REGION Network 37: [Spare_3] valve logic
   // Setup  //  Parametrierungshinweise
   // I_OpModeOutput  -->
   // 0=I_AutoOn schaltet den Ausgang Ein und Aus; 1=I_AutoOn schaltet ein und I_AutoAus schaltet aus
   // 0=I_AutoOn switches on and off; 1=I_AutoOn switches on and I_AutoOff switches off
   // 
   // I_OpModeAutoManual -->
   // 0=Automatik; 1=Hand
   // 0=Automatic; 1=Manual
   // 
   // I_AutoOn -->
   // 1=Automatik Ein, Eingang für die normalen Ventilverschaltungsbedingungen
   // 1=Automatic On, Input for the normal valve conditions
   // 
   // I_Release -->
   // 1=Freigabe, Eingang für die Fehlerbedingungen
   // 1=Release, Input for fault conditions
   // 
   // I_SafetyRelease -->
   // 1=Sicherheitsfreigabe, Eingang für zusätzliche Schaltbefehle aus dem Sicherheitsprogramm
   // 1=Safety release, Input for additional safety conditions from the safety program
   RUNG wire#powerrail
      Move(in := 0, out1 => "DB_R134a_BU_Values".Valve.Spare_3.Input.OpModeOutput)
      Move(in := "DB_R134a_AT_2_Values".OperationMode.ManualValveControl, out1 => "DB_R134a_BU_Values".Valve.Spare_3.Input.OpModeAutoManual)
      { S7_Templates := "SrcType := Int" } EQ_Contact(in1 := "DB_R134a_BU_Values".Valve.Spare_3.Input.OpModeAutoManual, in2 := 0)
      R_Coil( "DB_R134a_BU_Values".Valve.Spare_3.Input.ManualOn )
   END_RUNG
   RUNG wire#powerrail
      Contact( #Tmp_EnableOperation )
      Contact( "AlwaysFALSE" )
      Coil( "DB_R134a_BU_Values".Valve.Spare_3.Input.AutoOn )
   END_RUNG
   RUNG wire#powerrail
      Coil( "DB_R134a_BU_Values".Valve.Spare_3.Input.Release )
   END_RUNG
   RUNG wire#powerrail
      Coil( "DB_R134a_BU_Values".Valve.Spare_3.Input.SafetyRelease )
   END_RUNG
   RUNG wire#powerrail
      MOVE_BLK_VARIANT(SRC := "DB_R134a_1_StepData".Valve[1].Language, COUNT := 4, SRC_INDEX := 0, DEST_INDEX := 0, Ret_Val => #Tmp_ReturnValue, DEST => "DB_R134a_BU_Values".Valve.Spare_3.Input.TextName_Language)
   END_RUNG
   // the same network as SCL:
   "DB_R134a_BU_Values".Valve.Spare_3.Input.OpModeOutput := 0;
   "DB_R134a_BU_Values".Valve.Spare_3.Input.OpModeAutoManual := "DB_R134a_AT_2_Values".OperationMode.ManualValveControl;
   IF "DB_R134a_BU_Values".Valve.Spare_3.Input.OpModeAutoManual = 0 THEN
       "DB_R134a_BU_Values".Valve.Spare_3.Input.ManualOn := FALSE;
   END_IF;
   "DB_R134a_BU_Values".Valve.Spare_3.Input.AutoOn := #Tmp_EnableOperation AND "AlwaysFALSE";
   "DB_R134a_BU_Values".Valve.Spare_3.Input.Release := TRUE;
   "DB_R134a_BU_Values".Valve.Spare_3.Input.SafetyRelease := TRUE;
   #Tmp_ReturnValue := MOVE_BLK_VARIANT(SRC := "DB_R134a_1_StepData".Valve[1].Language,
                           COUNT := 4,
                           SRC_INDEX := 0,
                           DEST_INDEX := 0,
                           DEST => "DB_R134a_BU_Values".Valve.Spare_3.Input.TextName_Language);
END_REGION

REGION Network 38: [Spare_3] valve 1KM1VI1KKP11KKR14 - xxx.. - spare // Reserve
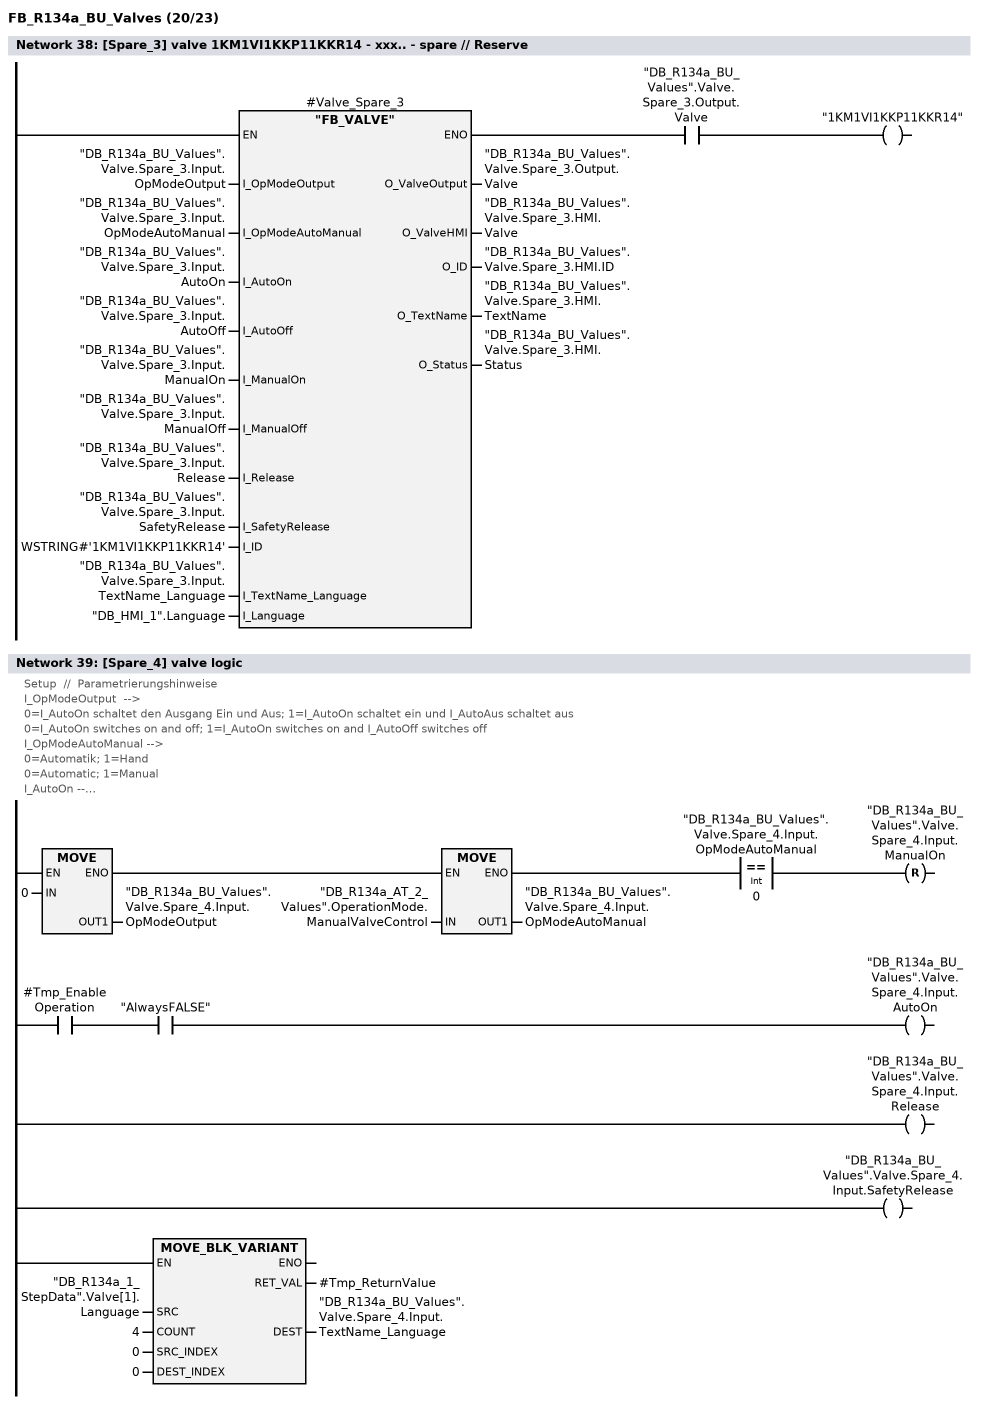
   RUNG wire#powerrail
      #Valve_Spare_3(I_OpModeOutput := "DB_R134a_BU_Values".Valve.Spare_3.Input.OpModeOutput, I_OpModeAutoManual := "DB_R134a_BU_Values".Valve.Spare_3.Input.OpModeAutoManual, I_AutoOn := "DB_R134a_BU_Values".Valve.Spare_3.Input.AutoOn, I_AutoOff := "DB_R134a_BU_Values".Valve.Spare_3.Input.AutoOff, I_ManualOn := "DB_R134a_BU_Values".Valve.Spare_3.Input.ManualOn, I_ManualOff := "DB_R134a_BU_Values".Valve.Spare_3.Input.ManualOff, I_Release := "DB_R134a_BU_Values".Valve.Spare_3.Input.Release, I_SafetyRelease := "DB_R134a_BU_Values".Valve.Spare_3.Input.SafetyRelease, I_ID := WSTRING#'1KM1VI1KKP11KKR14', I_TextName_Language := "DB_R134a_BU_Values".Valve.Spare_3.Input.TextName_Language, I_Language := "DB_HMI_1".Language, O_ValveOutput => "DB_R134a_BU_Values".Valve.Spare_3.Output.Valve, O_ValveHMI => "DB_R134a_BU_Values".Valve.Spare_3.HMI.Valve, O_ID => "DB_R134a_BU_Values".Valve.Spare_3.HMI.ID, O_TextName => "DB_R134a_BU_Values".Valve.Spare_3.HMI.TextName, O_Status => "DB_R134a_BU_Values".Valve.Spare_3.HMI.Status)
      Contact( "DB_R134a_BU_Values".Valve.Spare_3.Output.Valve )
      Coil( "1KM1VI1KKP11KKR14" )
   END_RUNG
   // the same network as SCL:
   #Valve_Spare_3(I_OpModeOutput := "DB_R134a_BU_Values".Valve.Spare_3.Input.OpModeOutput,   // "FB_VALVE"
                  I_OpModeAutoManual := "DB_R134a_BU_Values".Valve.Spare_3.Input.OpModeAutoManual,
                  I_AutoOn := "DB_R134a_BU_Values".Valve.Spare_3.Input.AutoOn,
                  I_AutoOff := "DB_R134a_BU_Values".Valve.Spare_3.Input.AutoOff,
                  I_ManualOn := "DB_R134a_BU_Values".Valve.Spare_3.Input.ManualOn,
                  I_ManualOff := "DB_R134a_BU_Values".Valve.Spare_3.Input.ManualOff,
                  I_Release := "DB_R134a_BU_Values".Valve.Spare_3.Input.Release,
                  I_SafetyRelease := "DB_R134a_BU_Values".Valve.Spare_3.Input.SafetyRelease,
                  I_ID := WSTRING#'1KM1VI1KKP11KKR14',
                  I_TextName_Language := "DB_R134a_BU_Values".Valve.Spare_3.Input.TextName_Language,
                  I_Language := "DB_HMI_1".Language,
                  O_ValveOutput => "DB_R134a_BU_Values".Valve.Spare_3.Output.Valve,
                  O_ValveHMI => "DB_R134a_BU_Values".Valve.Spare_3.HMI.Valve,
                  O_ID => "DB_R134a_BU_Values".Valve.Spare_3.HMI.ID,
                  O_TextName => "DB_R134a_BU_Values".Valve.Spare_3.HMI.TextName,
                  O_Status => "DB_R134a_BU_Values".Valve.Spare_3.HMI.Status,
                  ENO => #_w1);
   "1KM1VI1KKP11KKR14" := #_w1 AND "DB_R134a_BU_Values".Valve.Spare_3.Output.Valve;
END_REGION

REGION Network 39: [Spare_4] valve logic
   // Setup  //  Parametrierungshinweise
   // I_OpModeOutput  -->
   // 0=I_AutoOn schaltet den Ausgang Ein und Aus; 1=I_AutoOn schaltet ein und I_AutoAus schaltet aus
   // 0=I_AutoOn switches on and off; 1=I_AutoOn switches on and I_AutoOff switches off
   // 
   // I_OpModeAutoManual -->
   // 0=Automatik; 1=Hand
   // 0=Automatic; 1=Manual
   // 
   // I_AutoOn -->
   // 1=Automatik Ein, Eingang für die normalen Ventilverschaltungsbedingungen
   // 1=Automatic On, Input for the normal valve conditions
   // 
   // I_Release -->
   // 1=Freigabe, Eingang für die Fehlerbedingungen
   // 1=Release, Input for fault conditions
   // 
   // I_SafetyRelease -->
   // 1=Sicherheitsfreigabe, Eingang für zusätzliche Schaltbefehle aus dem Sicherheitsprogramm
   // 1=Safety release, Input for additional safety conditions from the safety program
   RUNG wire#powerrail
      Move(in := 0, out1 => "DB_R134a_BU_Values".Valve.Spare_4.Input.OpModeOutput)
      Move(in := "DB_R134a_AT_2_Values".OperationMode.ManualValveControl, out1 => "DB_R134a_BU_Values".Valve.Spare_4.Input.OpModeAutoManual)
      { S7_Templates := "SrcType := Int" } EQ_Contact(in1 := "DB_R134a_BU_Values".Valve.Spare_4.Input.OpModeAutoManual, in2 := 0)
      R_Coil( "DB_R134a_BU_Values".Valve.Spare_4.Input.ManualOn )
   END_RUNG
   RUNG wire#powerrail
      Contact( #Tmp_EnableOperation )
      Contact( "AlwaysFALSE" )
      Coil( "DB_R134a_BU_Values".Valve.Spare_4.Input.AutoOn )
   END_RUNG
   RUNG wire#powerrail
      Coil( "DB_R134a_BU_Values".Valve.Spare_4.Input.Release )
   END_RUNG
   RUNG wire#powerrail
      Coil( "DB_R134a_BU_Values".Valve.Spare_4.Input.SafetyRelease )
   END_RUNG
   RUNG wire#powerrail
      MOVE_BLK_VARIANT(SRC := "DB_R134a_1_StepData".Valve[1].Language, COUNT := 4, SRC_INDEX := 0, DEST_INDEX := 0, Ret_Val => #Tmp_ReturnValue, DEST => "DB_R134a_BU_Values".Valve.Spare_4.Input.TextName_Language)
   END_RUNG
   // the same network as SCL:
   "DB_R134a_BU_Values".Valve.Spare_4.Input.OpModeOutput := 0;
   "DB_R134a_BU_Values".Valve.Spare_4.Input.OpModeAutoManual := "DB_R134a_AT_2_Values".OperationMode.ManualValveControl;
   IF "DB_R134a_BU_Values".Valve.Spare_4.Input.OpModeAutoManual = 0 THEN
       "DB_R134a_BU_Values".Valve.Spare_4.Input.ManualOn := FALSE;
   END_IF;
   "DB_R134a_BU_Values".Valve.Spare_4.Input.AutoOn := #Tmp_EnableOperation AND "AlwaysFALSE";
   "DB_R134a_BU_Values".Valve.Spare_4.Input.Release := TRUE;
   "DB_R134a_BU_Values".Valve.Spare_4.Input.SafetyRelease := TRUE;
   #Tmp_ReturnValue := MOVE_BLK_VARIANT(SRC := "DB_R134a_1_StepData".Valve[1].Language,
                           COUNT := 4,
                           SRC_INDEX := 0,
                           DEST_INDEX := 0,
                           DEST => "DB_R134a_BU_Values".Valve.Spare_4.Input.TextName_Language);
END_REGION

REGION Network 40: [Spare_4] valve 1KM1VI1KKP11KKR12 - xxx.. - spare // Reserve
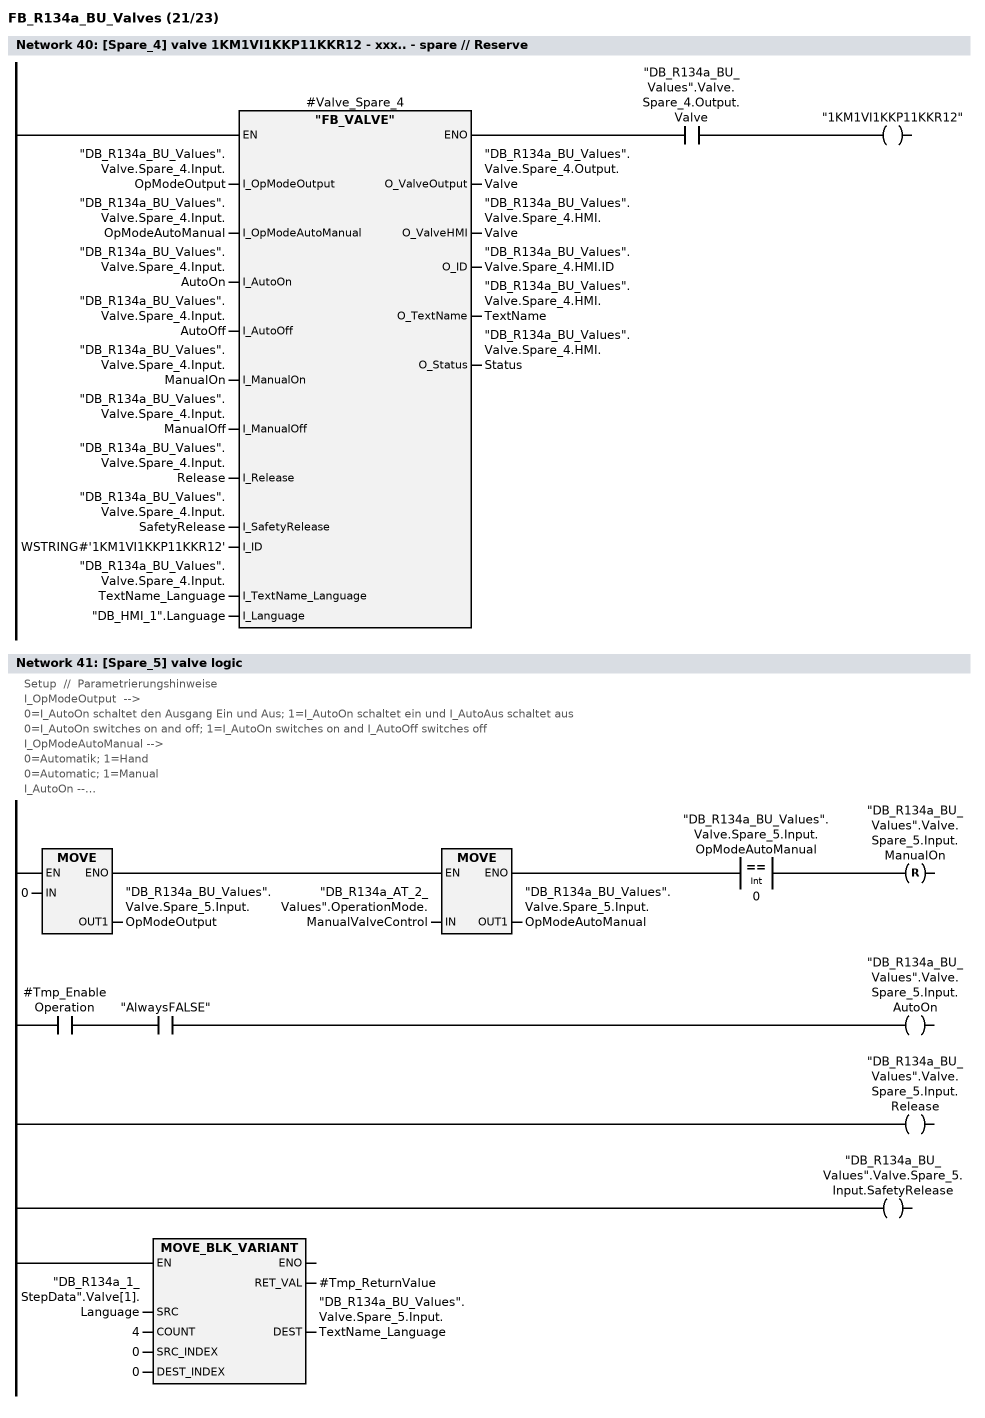
   RUNG wire#powerrail
      #Valve_Spare_4(I_OpModeOutput := "DB_R134a_BU_Values".Valve.Spare_4.Input.OpModeOutput, I_OpModeAutoManual := "DB_R134a_BU_Values".Valve.Spare_4.Input.OpModeAutoManual, I_AutoOn := "DB_R134a_BU_Values".Valve.Spare_4.Input.AutoOn, I_AutoOff := "DB_R134a_BU_Values".Valve.Spare_4.Input.AutoOff, I_ManualOn := "DB_R134a_BU_Values".Valve.Spare_4.Input.ManualOn, I_ManualOff := "DB_R134a_BU_Values".Valve.Spare_4.Input.ManualOff, I_Release := "DB_R134a_BU_Values".Valve.Spare_4.Input.Release, I_SafetyRelease := "DB_R134a_BU_Values".Valve.Spare_4.Input.SafetyRelease, I_ID := WSTRING#'1KM1VI1KKP11KKR12', I_TextName_Language := "DB_R134a_BU_Values".Valve.Spare_4.Input.TextName_Language, I_Language := "DB_HMI_1".Language, O_ValveOutput => "DB_R134a_BU_Values".Valve.Spare_4.Output.Valve, O_ValveHMI => "DB_R134a_BU_Values".Valve.Spare_4.HMI.Valve, O_ID => "DB_R134a_BU_Values".Valve.Spare_4.HMI.ID, O_TextName => "DB_R134a_BU_Values".Valve.Spare_4.HMI.TextName, O_Status => "DB_R134a_BU_Values".Valve.Spare_4.HMI.Status)
      Contact( "DB_R134a_BU_Values".Valve.Spare_4.Output.Valve )
      Coil( "1KM1VI1KKP11KKR12" )
   END_RUNG
   // the same network as SCL:
   #Valve_Spare_4(I_OpModeOutput := "DB_R134a_BU_Values".Valve.Spare_4.Input.OpModeOutput,   // "FB_VALVE"
                  I_OpModeAutoManual := "DB_R134a_BU_Values".Valve.Spare_4.Input.OpModeAutoManual,
                  I_AutoOn := "DB_R134a_BU_Values".Valve.Spare_4.Input.AutoOn,
                  I_AutoOff := "DB_R134a_BU_Values".Valve.Spare_4.Input.AutoOff,
                  I_ManualOn := "DB_R134a_BU_Values".Valve.Spare_4.Input.ManualOn,
                  I_ManualOff := "DB_R134a_BU_Values".Valve.Spare_4.Input.ManualOff,
                  I_Release := "DB_R134a_BU_Values".Valve.Spare_4.Input.Release,
                  I_SafetyRelease := "DB_R134a_BU_Values".Valve.Spare_4.Input.SafetyRelease,
                  I_ID := WSTRING#'1KM1VI1KKP11KKR12',
                  I_TextName_Language := "DB_R134a_BU_Values".Valve.Spare_4.Input.TextName_Language,
                  I_Language := "DB_HMI_1".Language,
                  O_ValveOutput => "DB_R134a_BU_Values".Valve.Spare_4.Output.Valve,
                  O_ValveHMI => "DB_R134a_BU_Values".Valve.Spare_4.HMI.Valve,
                  O_ID => "DB_R134a_BU_Values".Valve.Spare_4.HMI.ID,
                  O_TextName => "DB_R134a_BU_Values".Valve.Spare_4.HMI.TextName,
                  O_Status => "DB_R134a_BU_Values".Valve.Spare_4.HMI.Status,
                  ENO => #_w1);
   "1KM1VI1KKP11KKR12" := #_w1 AND "DB_R134a_BU_Values".Valve.Spare_4.Output.Valve;
END_REGION

REGION Network 41: [Spare_5] valve logic
   // Setup  //  Parametrierungshinweise
   // I_OpModeOutput  -->
   // 0=I_AutoOn schaltet den Ausgang Ein und Aus; 1=I_AutoOn schaltet ein und I_AutoAus schaltet aus
   // 0=I_AutoOn switches on and off; 1=I_AutoOn switches on and I_AutoOff switches off
   // 
   // I_OpModeAutoManual -->
   // 0=Automatik; 1=Hand
   // 0=Automatic; 1=Manual
   // 
   // I_AutoOn -->
   // 1=Automatik Ein, Eingang für die normalen Ventilverschaltungsbedingungen
   // 1=Automatic On, Input for the normal valve conditions
   // 
   // I_Release -->
   // 1=Freigabe, Eingang für die Fehlerbedingungen
   // 1=Release, Input for fault conditions
   // 
   // I_SafetyRelease -->
   // 1=Sicherheitsfreigabe, Eingang für zusätzliche Schaltbefehle aus dem Sicherheitsprogramm
   // 1=Safety release, Input for additional safety conditions from the safety program
   RUNG wire#powerrail
      Move(in := 0, out1 => "DB_R134a_BU_Values".Valve.Spare_5.Input.OpModeOutput)
      Move(in := "DB_R134a_AT_2_Values".OperationMode.ManualValveControl, out1 => "DB_R134a_BU_Values".Valve.Spare_5.Input.OpModeAutoManual)
      { S7_Templates := "SrcType := Int" } EQ_Contact(in1 := "DB_R134a_BU_Values".Valve.Spare_5.Input.OpModeAutoManual, in2 := 0)
      R_Coil( "DB_R134a_BU_Values".Valve.Spare_5.Input.ManualOn )
   END_RUNG
   RUNG wire#powerrail
      Contact( #Tmp_EnableOperation )
      Contact( "AlwaysFALSE" )
      Coil( "DB_R134a_BU_Values".Valve.Spare_5.Input.AutoOn )
   END_RUNG
   RUNG wire#powerrail
      Coil( "DB_R134a_BU_Values".Valve.Spare_5.Input.Release )
   END_RUNG
   RUNG wire#powerrail
      Coil( "DB_R134a_BU_Values".Valve.Spare_5.Input.SafetyRelease )
   END_RUNG
   RUNG wire#powerrail
      MOVE_BLK_VARIANT(SRC := "DB_R134a_1_StepData".Valve[1].Language, COUNT := 4, SRC_INDEX := 0, DEST_INDEX := 0, Ret_Val => #Tmp_ReturnValue, DEST => "DB_R134a_BU_Values".Valve.Spare_5.Input.TextName_Language)
   END_RUNG
   // the same network as SCL:
   "DB_R134a_BU_Values".Valve.Spare_5.Input.OpModeOutput := 0;
   "DB_R134a_BU_Values".Valve.Spare_5.Input.OpModeAutoManual := "DB_R134a_AT_2_Values".OperationMode.ManualValveControl;
   IF "DB_R134a_BU_Values".Valve.Spare_5.Input.OpModeAutoManual = 0 THEN
       "DB_R134a_BU_Values".Valve.Spare_5.Input.ManualOn := FALSE;
   END_IF;
   "DB_R134a_BU_Values".Valve.Spare_5.Input.AutoOn := #Tmp_EnableOperation AND "AlwaysFALSE";
   "DB_R134a_BU_Values".Valve.Spare_5.Input.Release := TRUE;
   "DB_R134a_BU_Values".Valve.Spare_5.Input.SafetyRelease := TRUE;
   #Tmp_ReturnValue := MOVE_BLK_VARIANT(SRC := "DB_R134a_1_StepData".Valve[1].Language,
                           COUNT := 4,
                           SRC_INDEX := 0,
                           DEST_INDEX := 0,
                           DEST => "DB_R134a_BU_Values".Valve.Spare_5.Input.TextName_Language);
END_REGION

REGION Network 42: [Spare_5] valve 1KM1VI1KKP12KKR14 - xxx.. - spare // Reserve
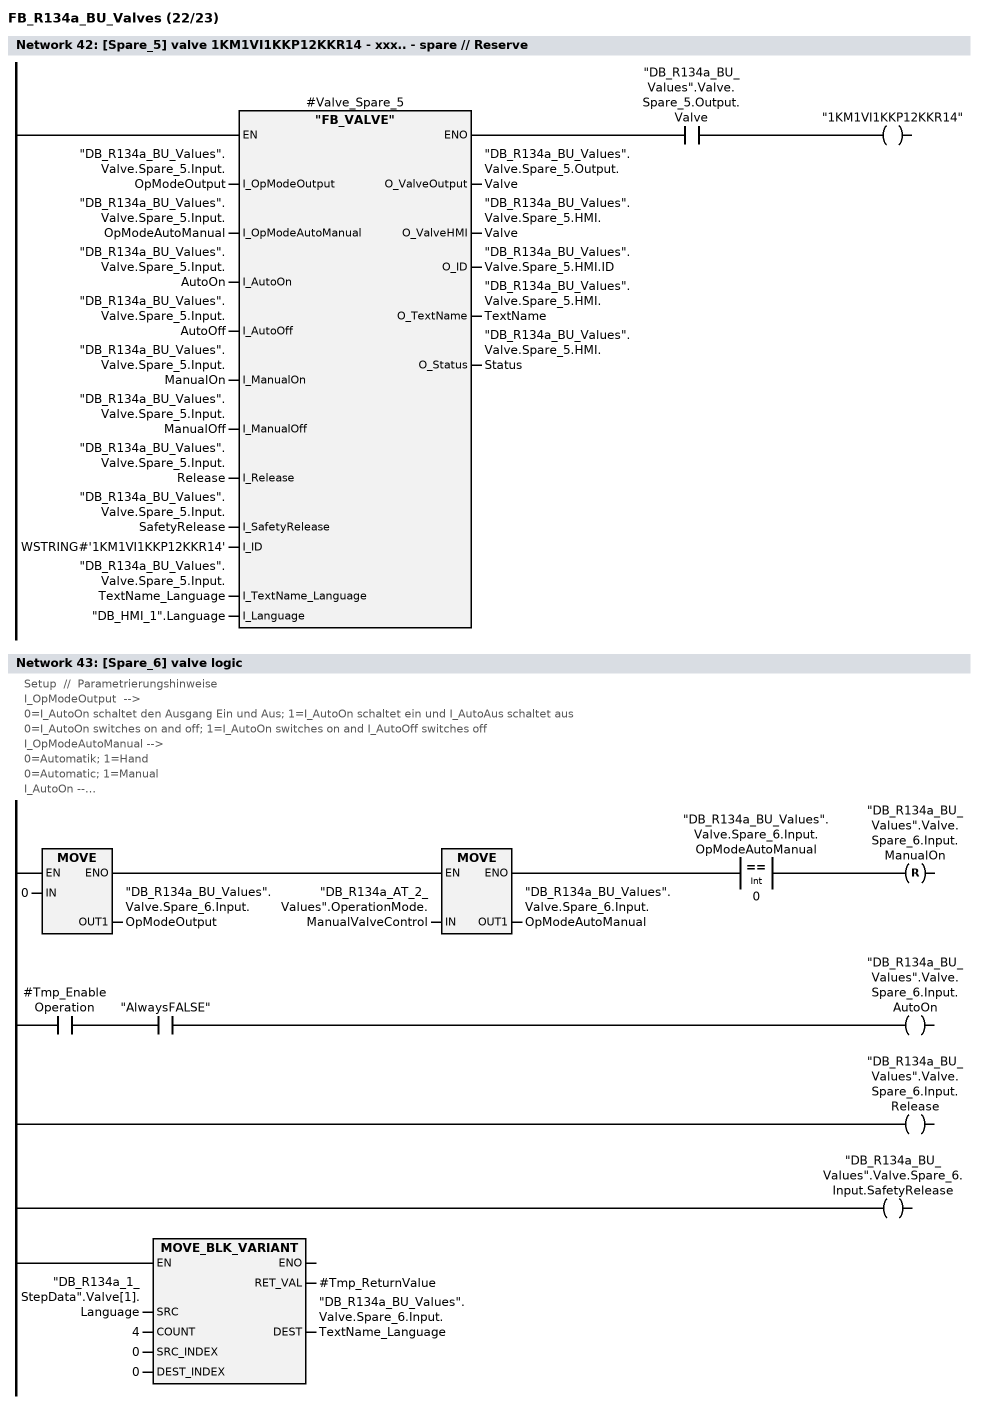
   RUNG wire#powerrail
      #Valve_Spare_5(I_OpModeOutput := "DB_R134a_BU_Values".Valve.Spare_5.Input.OpModeOutput, I_OpModeAutoManual := "DB_R134a_BU_Values".Valve.Spare_5.Input.OpModeAutoManual, I_AutoOn := "DB_R134a_BU_Values".Valve.Spare_5.Input.AutoOn, I_AutoOff := "DB_R134a_BU_Values".Valve.Spare_5.Input.AutoOff, I_ManualOn := "DB_R134a_BU_Values".Valve.Spare_5.Input.ManualOn, I_ManualOff := "DB_R134a_BU_Values".Valve.Spare_5.Input.ManualOff, I_Release := "DB_R134a_BU_Values".Valve.Spare_5.Input.Release, I_SafetyRelease := "DB_R134a_BU_Values".Valve.Spare_5.Input.SafetyRelease, I_ID := WSTRING#'1KM1VI1KKP12KKR14', I_TextName_Language := "DB_R134a_BU_Values".Valve.Spare_5.Input.TextName_Language, I_Language := "DB_HMI_1".Language, O_ValveOutput => "DB_R134a_BU_Values".Valve.Spare_5.Output.Valve, O_ValveHMI => "DB_R134a_BU_Values".Valve.Spare_5.HMI.Valve, O_ID => "DB_R134a_BU_Values".Valve.Spare_5.HMI.ID, O_TextName => "DB_R134a_BU_Values".Valve.Spare_5.HMI.TextName, O_Status => "DB_R134a_BU_Values".Valve.Spare_5.HMI.Status)
      Contact( "DB_R134a_BU_Values".Valve.Spare_5.Output.Valve )
      Coil( "1KM1VI1KKP12KKR14" )
   END_RUNG
   // the same network as SCL:
   #Valve_Spare_5(I_OpModeOutput := "DB_R134a_BU_Values".Valve.Spare_5.Input.OpModeOutput,   // "FB_VALVE"
                  I_OpModeAutoManual := "DB_R134a_BU_Values".Valve.Spare_5.Input.OpModeAutoManual,
                  I_AutoOn := "DB_R134a_BU_Values".Valve.Spare_5.Input.AutoOn,
                  I_AutoOff := "DB_R134a_BU_Values".Valve.Spare_5.Input.AutoOff,
                  I_ManualOn := "DB_R134a_BU_Values".Valve.Spare_5.Input.ManualOn,
                  I_ManualOff := "DB_R134a_BU_Values".Valve.Spare_5.Input.ManualOff,
                  I_Release := "DB_R134a_BU_Values".Valve.Spare_5.Input.Release,
                  I_SafetyRelease := "DB_R134a_BU_Values".Valve.Spare_5.Input.SafetyRelease,
                  I_ID := WSTRING#'1KM1VI1KKP12KKR14',
                  I_TextName_Language := "DB_R134a_BU_Values".Valve.Spare_5.Input.TextName_Language,
                  I_Language := "DB_HMI_1".Language,
                  O_ValveOutput => "DB_R134a_BU_Values".Valve.Spare_5.Output.Valve,
                  O_ValveHMI => "DB_R134a_BU_Values".Valve.Spare_5.HMI.Valve,
                  O_ID => "DB_R134a_BU_Values".Valve.Spare_5.HMI.ID,
                  O_TextName => "DB_R134a_BU_Values".Valve.Spare_5.HMI.TextName,
                  O_Status => "DB_R134a_BU_Values".Valve.Spare_5.HMI.Status,
                  ENO => #_w1);
   "1KM1VI1KKP12KKR14" := #_w1 AND "DB_R134a_BU_Values".Valve.Spare_5.Output.Valve;
END_REGION

REGION Network 43: [Spare_6] valve logic
   // Setup  //  Parametrierungshinweise
   // I_OpModeOutput  -->
   // 0=I_AutoOn schaltet den Ausgang Ein und Aus; 1=I_AutoOn schaltet ein und I_AutoAus schaltet aus
   // 0=I_AutoOn switches on and off; 1=I_AutoOn switches on and I_AutoOff switches off
   // 
   // I_OpModeAutoManual -->
   // 0=Automatik; 1=Hand
   // 0=Automatic; 1=Manual
   // 
   // I_AutoOn -->
   // 1=Automatik Ein, Eingang für die normalen Ventilverschaltungsbedingungen
   // 1=Automatic On, Input for the normal valve conditions
   // 
   // I_Release -->
   // 1=Freigabe, Eingang für die Fehlerbedingungen
   // 1=Release, Input for fault conditions
   // 
   // I_SafetyRelease -->
   // 1=Sicherheitsfreigabe, Eingang für zusätzliche Schaltbefehle aus dem Sicherheitsprogramm
   // 1=Safety release, Input for additional safety conditions from the safety program
   RUNG wire#powerrail
      Move(in := 0, out1 => "DB_R134a_BU_Values".Valve.Spare_6.Input.OpModeOutput)
      Move(in := "DB_R134a_AT_2_Values".OperationMode.ManualValveControl, out1 => "DB_R134a_BU_Values".Valve.Spare_6.Input.OpModeAutoManual)
      { S7_Templates := "SrcType := Int" } EQ_Contact(in1 := "DB_R134a_BU_Values".Valve.Spare_6.Input.OpModeAutoManual, in2 := 0)
      R_Coil( "DB_R134a_BU_Values".Valve.Spare_6.Input.ManualOn )
   END_RUNG
   RUNG wire#powerrail
      Contact( #Tmp_EnableOperation )
      Contact( "AlwaysFALSE" )
      Coil( "DB_R134a_BU_Values".Valve.Spare_6.Input.AutoOn )
   END_RUNG
   RUNG wire#powerrail
      Coil( "DB_R134a_BU_Values".Valve.Spare_6.Input.Release )
   END_RUNG
   RUNG wire#powerrail
      Coil( "DB_R134a_BU_Values".Valve.Spare_6.Input.SafetyRelease )
   END_RUNG
   RUNG wire#powerrail
      MOVE_BLK_VARIANT(SRC := "DB_R134a_1_StepData".Valve[1].Language, COUNT := 4, SRC_INDEX := 0, DEST_INDEX := 0, Ret_Val => #Tmp_ReturnValue, DEST => "DB_R134a_BU_Values".Valve.Spare_6.Input.TextName_Language)
   END_RUNG
   // the same network as SCL:
   "DB_R134a_BU_Values".Valve.Spare_6.Input.OpModeOutput := 0;
   "DB_R134a_BU_Values".Valve.Spare_6.Input.OpModeAutoManual := "DB_R134a_AT_2_Values".OperationMode.ManualValveControl;
   IF "DB_R134a_BU_Values".Valve.Spare_6.Input.OpModeAutoManual = 0 THEN
       "DB_R134a_BU_Values".Valve.Spare_6.Input.ManualOn := FALSE;
   END_IF;
   "DB_R134a_BU_Values".Valve.Spare_6.Input.AutoOn := #Tmp_EnableOperation AND "AlwaysFALSE";
   "DB_R134a_BU_Values".Valve.Spare_6.Input.Release := TRUE;
   "DB_R134a_BU_Values".Valve.Spare_6.Input.SafetyRelease := TRUE;
   #Tmp_ReturnValue := MOVE_BLK_VARIANT(SRC := "DB_R134a_1_StepData".Valve[1].Language,
                           COUNT := 4,
                           SRC_INDEX := 0,
                           DEST_INDEX := 0,
                           DEST => "DB_R134a_BU_Values".Valve.Spare_6.Input.TextName_Language);
END_REGION

REGION Network 44: [Spare_6] valve 1KM1VI1KKP12KKR12 - xxx.. - spare // Reserve
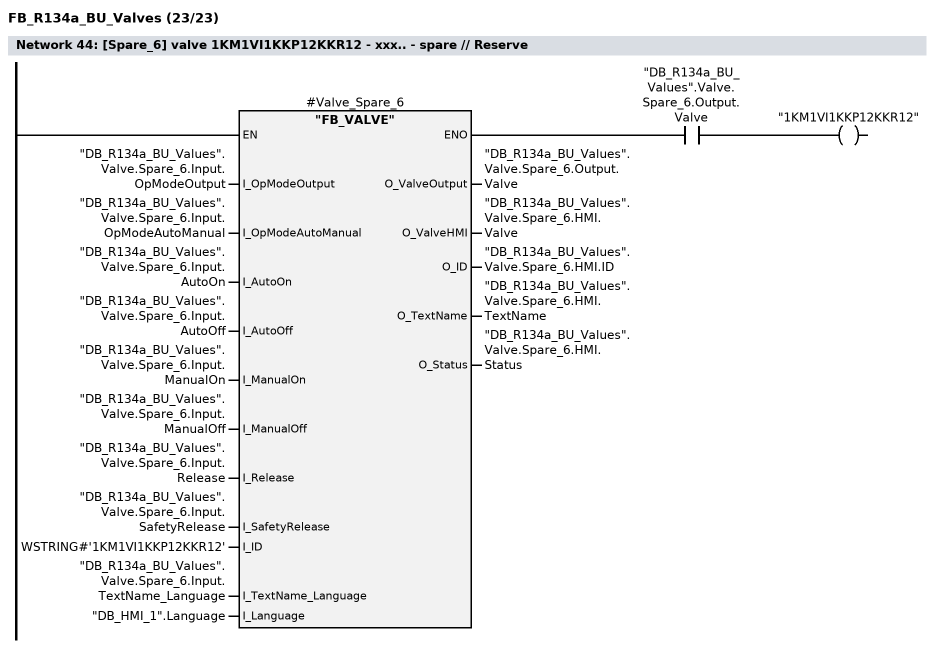
   RUNG wire#powerrail
      #Valve_Spare_6(I_OpModeOutput := "DB_R134a_BU_Values".Valve.Spare_6.Input.OpModeOutput, I_OpModeAutoManual := "DB_R134a_BU_Values".Valve.Spare_6.Input.OpModeAutoManual, I_AutoOn := "DB_R134a_BU_Values".Valve.Spare_6.Input.AutoOn, I_AutoOff := "DB_R134a_BU_Values".Valve.Spare_6.Input.AutoOff, I_ManualOn := "DB_R134a_BU_Values".Valve.Spare_6.Input.ManualOn, I_ManualOff := "DB_R134a_BU_Values".Valve.Spare_6.Input.ManualOff, I_Release := "DB_R134a_BU_Values".Valve.Spare_6.Input.Release, I_SafetyRelease := "DB_R134a_BU_Values".Valve.Spare_6.Input.SafetyRelease, I_ID := WSTRING#'1KM1VI1KKP12KKR12', I_TextName_Language := "DB_R134a_BU_Values".Valve.Spare_6.Input.TextName_Language, I_Language := "DB_HMI_1".Language, O_ValveOutput => "DB_R134a_BU_Values".Valve.Spare_6.Output.Valve, O_ValveHMI => "DB_R134a_BU_Values".Valve.Spare_6.HMI.Valve, O_ID => "DB_R134a_BU_Values".Valve.Spare_6.HMI.ID, O_TextName => "DB_R134a_BU_Values".Valve.Spare_6.HMI.TextName, O_Status => "DB_R134a_BU_Values".Valve.Spare_6.HMI.Status)
      Contact( "DB_R134a_BU_Values".Valve.Spare_6.Output.Valve )
      Coil( "1KM1VI1KKP12KKR12" )
   END_RUNG
   // the same network as SCL:
   #Valve_Spare_6(I_OpModeOutput := "DB_R134a_BU_Values".Valve.Spare_6.Input.OpModeOutput,   // "FB_VALVE"
                  I_OpModeAutoManual := "DB_R134a_BU_Values".Valve.Spare_6.Input.OpModeAutoManual,
                  I_AutoOn := "DB_R134a_BU_Values".Valve.Spare_6.Input.AutoOn,
                  I_AutoOff := "DB_R134a_BU_Values".Valve.Spare_6.Input.AutoOff,
                  I_ManualOn := "DB_R134a_BU_Values".Valve.Spare_6.Input.ManualOn,
                  I_ManualOff := "DB_R134a_BU_Values".Valve.Spare_6.Input.ManualOff,
                  I_Release := "DB_R134a_BU_Values".Valve.Spare_6.Input.Release,
                  I_SafetyRelease := "DB_R134a_BU_Values".Valve.Spare_6.Input.SafetyRelease,
                  I_ID := WSTRING#'1KM1VI1KKP12KKR12',
                  I_TextName_Language := "DB_R134a_BU_Values".Valve.Spare_6.Input.TextName_Language,
                  I_Language := "DB_HMI_1".Language,
                  O_ValveOutput => "DB_R134a_BU_Values".Valve.Spare_6.Output.Valve,
                  O_ValveHMI => "DB_R134a_BU_Values".Valve.Spare_6.HMI.Valve,
                  O_ID => "DB_R134a_BU_Values".Valve.Spare_6.HMI.ID,
                  O_TextName => "DB_R134a_BU_Values".Valve.Spare_6.HMI.TextName,
                  O_Status => "DB_R134a_BU_Values".Valve.Spare_6.HMI.Status,
                  ENO => #_w1);
   "1KM1VI1KKP12KKR12" := #_w1 AND "DB_R134a_BU_Values".Valve.Spare_6.Output.Valve;
END_REGION
END_FUNCTION_BLOCK
